Staubli VAL3: detection.pgx

program detection()
  local num l_i
  local num l_nObjDetected
  local num l_nNumOfPart
begin
  // This is a sample program for the detection library to be used
  // with VALTRACK software.
  //
  // Misc
  // You can use this program "as is" if your detection device is a sensor
  // in that case:
  // - you will detect only one single object (l_nNumOfPart=1)
  // - the object will have ID 1 (one)
  // - the coordinate of the object must be defined in your main application
  //
  // In case you have a camera, you should comment or erase the Sensor section
  // and use the camera section.
  // write your own routines to get the necessary data from the camera.
  //
  //----------------------------------------------------------------
  //
  // detection task running : unlock the task's conveyor when valtrack  begins
  bTaskDetOK=true
  //********** Sensor section
  do
    nObjectID[0]=1
    trObjectPos[0]={0,0,0,0,0,0}
    nNumOfPart=1
    wait(nNumOfPart==-1)
    delay(0)
  until false
  return
  //********** end of Sensor section
  //
  //********** Camera section
  //init cam
  // detection task running : unlock the task's conveyor when valtrack  begins
  //bTaskDetOK=true
  do
    // wait until camera has finished image treatment
    // call WaitUntilCameraReady()
    //
    // Read how many object have been detected.
    // Call myRoutineToReadNumberOfDetectedObject(l_nObjDetected)
    //
    l_nNumOfPart=0
    for l_i=0 to l_nObjDetected-1
      // Read data from your detection device:
      // Call myRoutineToReadObjectData (nObjectID[l_nNumOfPart],trObjectPos[l_nNumOfPart])
      //
      // increment l_nNumOfPart only if you want to bufferize the object.
      // For instance, you bufferize object only with:
      //        - ID=1
      //        - positive Y coordinate
      //
      //if (nObjectID[l_nNumOfPart]==1) and (trObjectPos[l_nNumOfPart].y)>0)
      //  l_nNumOfPart=l_nNumOfPart+1
      //endIf
    endFor
    //
    // Set number of detected parts.
    // nNumOfPart is watched by the conveyor library.
    //  Once nNumOfPart is set, the conveyor library will access
    //  the variables nObjectID[] and trObjectPos[].
    //  They must be fully updated before nNumOfPart is set.
    nNumOfPart=l_nNumOfPart
    //
    // Once data have been read by conveyor library
    // nNumOfPart is set to value -1
    wait(nNumOfPart==-1)
    //
    delay(0)
  until false
  //********** end of camera section
end
